ABB RAPID module: Module2023_real.mod

MODULE Module1
    	CONST robtarget Pos_origen:=[[324.49,-78.27,659.60],[0.0272456,0.994094,0.103028,-0.0205144],[-1,-1,1,0],[9E+09,9E+09,9E+09,9E+09,9E+09,9E+09]];
	CONST robtarget Pos_prepick_Brick:= [[303.02,-563.01,614.21],[0.0217975,-0.993749,-0.102158,0.0393898],[-1,-1,1,0],[9E+09,9E+09,9E+09,9E+09,9E+09,9E+09]];
	CONST robtarget Pos_pick_Brick:=    [[303.02,-563.01,492.30],[0.0217964,-0.993749,-0.102155,0.0393871],[-1,-1,1,0],[9E+09,9E+09,9E+09,9E+09,9E+09,9E+09]];
	CONST robtarget Pos_preplace_Brick:=[[450.22,-250.83,423.59],[0.000478151,-0.994466,-0.102418,0.0233921],[-1,-1,1,0],[9E+09,9E+09,9E+09,9E+09,9E+09,9E+09]];
	CONST robtarget Pos_place_Brick:=   [[450.22,-241.00,339.11],[0.000479484,-0.994467,-0.102415,0.0233942],[-1,-1,1,0],[9E+09,9E+09,9E+09,9E+09,9E+09,9E+09]];
	CONST robtarget Pos_prepick_lata:=  [[248.46,-547.24,580.87],[0.0217764,-0.993758,-0.102113,0.0392901],[-1,-1,1,0],[9E+09,9E+09,9E+09,9E+09,9E+09,9E+09]];
	CONST robtarget Pos_pick_lata:=     [[248.46,-547.24,503.07],[0.0217784,-0.993757,-0.10212,0.0392927],[-1,-1,1,0],[9E+09,9E+09,9E+09,9E+09,9E+09,9E+09]];
	CONST robtarget Pos_preplace_lata:= [[401.08,117.50,421.70],[0.0272257,0.994092,0.103046,-0.0205288],[0,-1,2,0],[9E+09,9E+09,9E+09,9E+09,9E+09,9E+09]];
	CONST robtarget Pos_place_lata:=    [[401.08,117.50,353.44],[0.0272261,0.994092,0.103042,-0.0205267],[0,-1,2,0],[9E+09,9E+09,9E+09,9E+09,9E+09,9E+09]];


    VAR robtarget prepick_var;
    VAR robtarget pick_var;
ENDMODULE
